FUNCTION F_SubstractFunction : REAL
VAR_INPUT
	rInput1 : REAL;
	rInput2 : REAL;
END_VAR
VAR
END_VAR

F_SubstractFunction := rInput1 - rInput2;

END_FUNCTION

(* stored: Version 1.1.0.1, ProductVersion 3.1.4024.13
   POU F_SubstractFunction: Id {a578b3b4-d4e5-49e9-a662-146f834fa651}, SpecialFunc None *)
